DATA_BLOCK "bioPID.D"
TITLE = Batch I/O PID Data Block
{ S7_Optimized_Access := 'TRUE' }
AUTHOR : Woermann
VERSION : 1.0
// -- Woermann Automation --
// Date: 2020-06-20
NON_RETAIN
   VAR RETAIN
      pid : Array[0..15] of "bioPID.DT";
   END_VAR

BEGIN

END_DATA_BLOCK

